FUNCTION_BLOCK FB_RobotAbsMove EXTENDS FB_ObjectBase_V2 IMPLEMENTS IBasicElement
VAR_INPUT
    Robot         : REFERENCE TO FB_FanucRobot_Basic_V2;
    LowerConveyor : REFERENCE TO FB_Motor;
    // Command   : ST_WareHouseWithRobotMove_Command;
    Info : st_AutoSixAxisAbsMoveParameter;
	Input :ST_InputTable;
    Stop : BOOL;
END_VAR
VAR_OUTPUT
    // Status : ST_WareHouseWithRobotMove_Status;
END_VAR
VAR
    _Abort       : BOOL;
    strStatus    : STRING;
    uiResumeStep : UINT;

    Area : E_RobotArea;
    UseA : BOOL;
    UseB : BOOL;

    Get                         : BOOL;
    tonTimeOut                  : TON;
	TON_DelayLowerCV			: TON;
    _UniqueErrorCode            : STRING;
    FirstSensorOfLowerConveyor  : BOOL;
    SecondSensorOfLowerConveyor : BOOL;

END_VAR

SUPER^.A10_StateControl();
A00_BasicUnits();
FirstSensorOfLowerConveyor := Input.bLowCV_BoxArrived_Sensor;
SecondSensorOfLowerConveyor := Input.bLowCV_2ndBoxGap_Sensor;

ACTION A00_BasicUnits:
tonTimeOut(PT:=T#60S);
TON_DelayLowerCV(PT:=T#1S);
ErrorID :=2200;
END_ACTION

METHOD M_CheckCommand : BOOL // True : Command is useful
VAR_INPUT
END_VAR
VAR
	
END_VAR
// Check command paremeter is correct


IF Info.A_Get <> Info.B_Get THEN
	strStatus:='Wrong command ,GetA not match to GetB';
	M_CheckCommand:=FALSE;
	RETURN;
ELSE		
	THIS^.Get :=Info.A_Get;
END_IF

IF Info.A_Area<> Info.B_Area THEN
	IF NOT(Info.A_Area=99 OR Info.B_Area=99) THEN
	strStatus:='Wrong command ,Area A not match to Area B';
	M_CheckCommand:=FALSE;
	RETURN;
END_IF
END_IF

IF Info.A_Area = 99 AND Info.B_Area = 99 THEN
	strStatus:='Wrong command ,Both Area are 99';
	M_CheckCommand:=FALSE;
	RETURN;
END_IF

CASE LREAL_TO_INT(Info.A_Area) OF
	1 : //Normal command : RoundBelt
		IF Info.A_Position<1 OR  Info.A_Position>3 THEN
			strStatus:='Wrong command ,Position A Not allow';
			M_CheckCommand:=FALSE;
			RETURN;	
		ELSE
			Area := E_RobotArea.RoundBelt;
			UseA :=TRUE	;	
		END_IF
		
	2:	//Buffer area
		IF Info.A_Position<1 OR  Info.A_Position>40 THEN
			strStatus:='Wrong command ,Position A Not allow';
			M_CheckCommand:=FALSE;
			RETURN;	
		ELSE
			Area := E_RobotArea.BufferArea;
			UseA :=TRUE	;	
		END_IF
	3: //Allocated/Empty conveyor
		IF Info.A_Position<1 OR  Info.A_Position>2 THEN
			strStatus:='Wrong command ,Position A Not allow';
			M_CheckCommand:=FALSE;
			RETURN;	
		ELSE
			Area := E_RobotArea.TransmitCV;
			UseA :=TRUE	;	
		END_IF
	5: //FeedIn/Out conveyor
		IF Info.A_Position<1 OR  Info.A_Position>3 THEN
			strStatus:='Wrong command ,Position A Not allow';
			M_CheckCommand:=FALSE;
			RETURN;	
		ELSIF Info.A_Position=3 AND Get THEN
			strStatus:='Wrong command ,Can Not Get box from FeedOut conveyor ';
			M_CheckCommand:=FALSE;
			RETURN;	
		ELSE
			Area := E_RobotArea.InOutConveyor;
			UseA :=TRUE	;	
		END_IF
	7: // PullOut conveyor
		IF Info.A_Position<1 OR  Info.A_Position>2 THEN
			strStatus:='Wrong command ,Position A Not allow';
			M_CheckCommand:=FALSE;
			RETURN;	
		ELSE
			Area := E_RobotArea.PullOutConveyor;
			UseA :=TRUE	;	
		END_IF
	
	99: //ClampA not use
		UseA :=FALSE;
	
	ELSE //Wrong command
		strStatus:='Wrong command ,Area_A not allow ';
		M_CheckCommand:=FALSE;
		RETURN;

END_CASE

CASE LREAL_TO_INT(Info.B_Area) OF
	1 : //Normal command : RoundBelt
		IF Info.B_Position<1 OR  Info.B_Position>3 THEN
			strStatus:='Wrong command ,Position B Not allow';
			M_CheckCommand:=FALSE;
			RETURN;	
		ELSE
			Area := E_RobotArea.RoundBelt;
			UseB :=TRUE	;	
		END_IF
		
	2:	
		IF Info.B_Position<1 OR  Info.B_Position>40 THEN
			strStatus:='Wrong command ,Position B Not allow';
			M_CheckCommand:=FALSE;
			RETURN;	
		ELSE
			Area := E_RobotArea.BufferArea;
			UseB :=TRUE	;	
		END_IF
	3:
		IF Info.B_Position<1 OR  Info.B_Position>2 THEN
			strStatus:='Wrong command ,Position B Not allow';
			M_CheckCommand:=FALSE;
			RETURN;	
		ELSE
			Area := E_RobotArea.TransmitCV;
			UseB :=TRUE	;	
		END_IF
	5:
		IF Info.B_Position<1 OR  Info.B_Position>3 THEN
			strStatus:='Wrong command ,Position B Not allow';
			M_CheckCommand:=FALSE;
			RETURN;	
		ELSE
			Area := E_RobotArea.InOutConveyor;
			UseB :=TRUE	;	
		END_IF
	7:
		IF Info.B_Position<1 OR  Info.B_Position>2 THEN
			strStatus:='Wrong command ,Position B Not allow';
			M_CheckCommand:=FALSE;
			RETURN;	
		ELSIF Info.B_Position=3 AND Get THEN
			strStatus:='Wrong command ,Can Not Get box from FeedOut conveyor ';
			M_CheckCommand:=FALSE;
			RETURN;	
		ELSE
			Area := E_RobotArea.PullOutConveyor;
			UseB :=TRUE	;	
		END_IF
	
	99: //ClampA not use
		UseB :=FALSE;
	
	ELSE //Wrong command
		strStatus:='Wrong command ,Area_B not allow ';
		M_CheckCommand:=FALSE;
		RETURN;

END_CASE


M_CheckCommand:=TRUE;
END_METHOD

METHOD M_CheckUnitsNotBusy : BOOL
VAR_INPUT
END_VAR
M_CheckUnitsNotBusy := true;
END_METHOD

METHOD M_CheckUnitsReady : BOOL
VAR_INPUT
END_VAR
M_CheckUnitsReady := true;
END_METHOD

METHOD  M_STATE_ABORTED
VAR_INPUT
END_VAR
ERROR :=TRUE;
Busy    := FALSE;
Aborted := TRUE;
Status := strStatus;
UniqueErrorCode:=_UniqueErrorCode;
IF NOT Execute THEN
	eSTATE:=STATE_RESETTING;
END_IF

IF Execute AND Reset THEN
	uiExecutingStep :=uiResumeStep;
	eSTATE:=STATE_EXECUTING;
END_IF
END_METHOD

METHOD  M_STATE_ABORTING
VAR_INPUT
END_VAR
CASE uiAbortingStep OF
	0 :
		uiAbortingStep:=9999;
	
	9999:	_AbortCompleted:=TRUE;
END_CASE

IF _AbortCompleted THEN	
	eSTATE :=STATE_ABORTED;
END_IF
END_METHOD

METHOD  M_STATE_DONE
VAR_INPUT
END_VAR
Busy := FALSE;
Done := TRUE;
IF NOT Execute THEN
    eState := STATE_RESETTING;
END_IF
END_METHOD

METHOD  M_STATE_DORMANT
VAR_INPUT
END_VAR
// Clear FB output
Busy            := FALSE;
Done            := FALSE;
Aborted         := FALSE;
Error           := FALSE;
ErrorID         := 0;
Status          := '';
_ResetCompleted := FALSE;
_Error          := FALSE;
_Executed       := FALSE;

tonTimeOut.IN:=FALSE;
TON_DelayLowerCV.IN := false;
strStatus :='No Error';
uiExecutingStep :=uiResettingStep :=uiResumeStep :=0;


// Wait Execute command
IF Execute THEN
    eState := STATE_EXECUTING;
END_IF
END_METHOD

METHOD  M_STATE_ERROR
VAR_INPUT
END_VAR
ERROR   :=TRUE;
Busy	:=FALSE;
Status := strStatus;
UniqueErrorCode:=_UniqueErrorCode;
ErrorID :=2200;
IF NOT Execute THEN	
eSTATE:=STATE_RESETTING;
END_IF
END_METHOD

METHOD  M_STATE_EXECUTING
VAR_INPUT
END_VAR
VAR_INST
    ActionMode       : E_ReloadRoundBoxAction;
	BoxReady_1st : BOOL;
	BoxReady_2nd : BOOL;
    CarrierReady_1st : BOOL;
    CarrierReady_2nd : BOOL;
    uiBothStep : UINT;
    uiSingleClampStep : UINT;	
	Area : E_RobotArea;
	Address_A : INT;
	Address_B : INT;
END_VAR
VAR
	WareHouse: INT;
END_VAR
// Set Busy active edit by johnson
Busy := TRUE;
IF THIS^.Stop THEN // Pending the timeout when Stop signal occur
	tonTimeout.IN :=FALSE;
END_IF
// Service Process
CASE uiExecutingStep OF
	0:
        // Clear variable
        ActionMode       := E_ReloadRoundBoxAction.Undefined;
        CarrierReady_1st := FALSE;
        CarrierReady_2nd := FALSE;
        uiBothStep := 0;
		uiSingleClampStep :=0;
		BoxReady_1st := 0;
		BoxReady_2nd := 0;
		tonTimeOut.IN:=FALSE;
        // Check command
        IF M_CheckCommand() THEN
            uiExecutingStep := 10;
		ELSE
			_Error:=TRUE;
        END_IF
    10:
        // Start process, check units first
        IF M_CheckUnitsReady() THEN
            uiExecutingStep := 20;
        END_IF
    20:
        // CHeck units not busy state
        IF M_CheckUnitsNotBusy() THEN
            uiExecutingStep := 1000;
        END_IF
   
	1000:   
			// Read   coordinate
			 Area := THIS^.Area;
 			 Address_A := LREAL_TO_INT(Info.A_Position);
			 Address_B := LREAL_TO_INT(Info.B_Position);
			 
			IF UseA AND NOT UseB THEN
				//Only clampA
				uiExecutingStep := 10000;
			ELSIF NOT UseA AND UseB THEN
				//Only ClampB 
				uiExecutingStep := 20000;
			ELSIF UseA AND UseB THEN
				//Both Clamps
				uiExecutingStep := 30000;		
			END_IF
       
    10000: // Only ClampA 
        IF NOT Robot._DI1.Done THEN
            
            
			CASE uiSingleClampStep OF
				
				0://
					IF Area= E_RobotArea.InOutConveyor AND Address_A=3 THEN
						uiSingleClampStep:=100;// Need to control feedout conveyor 
					ELSE
						uiSingleClampStep:=1000;	
					END_IF
				100:	//check the box is full 
					IF Input.bLowCV_Block2Detect_Sensor THEN 
						_Error := TRUE;
						strStatus :='LowerCV the box behind is full, please remove it';
					ELSE 
						uiSingleClampStep := 150;
					END_IF
				
				150:	//check the box not no the  sensor 
					IF  FirstSensorOfLowerConveyor OR  (NOT SecondSensorOfLowerConveyor) THEN
						LowerConveyor.M_MoveBackward();
						tonTimeOut.IN:=FALSE;;
						uiSingleClampStep:=200;
					ELSE 
						uiSingleClampStep := 1000;
					END_IF
					tonTimeOut.IN:=TRUE;
					IF tonTimeOut.Q=TRUE THEN
						strStatus :='Empty Conveyor timeout';
						_Error:=TRUE;
					END_IF
				200:
//					TON_DelayLowerCV.IN := TRUE;
//					IF TON_DelayLowerCV.Q THEN
//					LowerConveyor.M_MotorStop();
//					uiSingleClampStep:=300;
//					END_IF 
					IF Input.bLowCV_Block2Detect_Sensor THEN
						TON_DelayLowerCV.IN := TRUE;
					END_IF
					IF TON_DelayLowerCV.Q THEN
						LowerConveyor.M_MotorStop();
						uiSingleClampStep := 300;
					END_IF
									
				300:
					TON_DelayLowerCV.IN :=FALSE;
					IF 	LowerConveyor.InStopped THEN
						tonTimeOut.IN:=FALSE;
						uiSingleClampStep:=1000;
					END_IF
					tonTimeOut.IN:=TRUE;
					IF tonTimeOut.Q=TRUE THEN
						strStatus :='Stop Conveyor timeout';
						_Error:=TRUE;
					END_IF	
				1000:
						BoxReady_1st:=TRUE;
						uiSingleClampStep:=9999;
				9999: //Wait	
			END_CASE
			          		 
				  // Robot Abs move
           		 Robot.M_StartRobotAbsMove(GetBox:=Get,
											UseClampA:=UseA,
											UseClampB:=UseB,
											Area:=Area,
											ClampA_Address:=Address_A,
											ClampB_Address:=Address_B,
											BoxReady_1:=BoxReady_1st,
											BoxReady_2:=BoxReady_2nd);				  
		
        ELSE
            uiExecutingStep := 10080;
        END_IF
		
    10080:
        Robot.M_ResetRobotAbsMove(UseA,UseB); // Clear command and go to place box
		tonTimeOut.IN:=TRUE;
        IF NOT Robot._DI1.Done THEN
			tonTimeOut.IN:=FALSE;
            uiExecutingStep := 40000; 
        END_IF
    	IF tonTimeOut.Q=TRUE THEN
			strStatus :='Reset Robot timeout';
			_Error:=TRUE;
		END_IF
		
    
   20000: // Only ClampB
        IF NOT Robot._DI1.Done THEN
            			
			CASE uiSingleClampStep OF
				
				0://
					IF Area= E_RobotArea.InOutConveyor AND Address_B=3 THEN
						uiSingleClampStep:=100;// Need to control feedout conveyor 
					ELSE
						uiSingleClampStep:=1000;	
					END_IF
					
				100:	//check the box is full 
					IF Input.bLowCV_Block2Detect_Sensor THEN 
						_Error := TRUE;
						strStatus :='LowerCV the box behind is full, please remove it';
					ELSE 
						uiSingleClampStep := 150;
					END_IF
				
				150:	//check the box not no the  sensor 
					IF  FirstSensorOfLowerConveyor OR  (NOT SecondSensorOfLowerConveyor) THEN
						LowerConveyor.M_MoveBackward();
						tonTimeOut.IN:=FALSE;;
						uiSingleClampStep:=200;
					ELSE
						uiSingleClampStep := 1000;
					END_IF
					tonTimeOut.IN:=TRUE;
					IF tonTimeOut.Q=TRUE THEN
						strStatus :='Empty Conveyor timeout';
						_Error:=TRUE;
					END_IF
				200:
//					TON_DelayLowerCV.IN := TRUE;
//					IF TON_DelayLowerCV.Q THEN
//					LowerConveyor.M_MotorStop();
//					uiSingleClampStep:=300;
//					END_IF 
					IF Input.bLowCV_Block2Detect_Sensor THEN
						TON_DelayLowerCV.IN := TRUE;
					END_IF
					IF TON_DelayLowerCV.Q THEN
						LowerConveyor.M_MotorStop();
						uiSingleClampStep := 300;
					END_IF
									
				300:
					TON_DelayLowerCV.IN :=FALSE;
					IF 	LowerConveyor.InStopped THEN
						tonTimeOut.IN:=FALSE;
						uiSingleClampStep:=1000;
					END_IF
					tonTimeOut.IN:=TRUE;
					IF tonTimeOut.Q=TRUE THEN
						strStatus :='Stop Conveyor timeout';
						_Error:=TRUE;
					END_IF	
				1000:
						BoxReady_2nd:=TRUE;
						uiSingleClampStep:=9999;
				9999: //Wait			
			END_CASE
			          		 
				  // Robot Abs move
           		 Robot.M_StartRobotAbsMove( GetBox:=Get,
											UseClampA:=UseA,
											UseClampB:=UseB,
											Area:=Area,
											ClampA_Address:=Address_A,
											ClampB_Address:=Address_B,
											BoxReady_1:=BoxReady_1st,
											BoxReady_2:=BoxReady_2nd);	
        ELSE
            uiExecutingStep := 20080;
        END_IF
		
    20080:
       Robot.M_ResetRobotAbsMove(UseA,UseB);; // Clear command 

        IF NOT Robot._DI1.Done THEN
            uiExecutingStep := 40000; 
        END_IF
		tonTimeOut.IN:=TRUE;
		IF tonTimeOut.Q=TRUE THEN
			strStatus :='Reset Robot timeout';
			_Error:=TRUE;
		END_IF	
    30000: // Both Clamps
        		
		
		  CASE uiBothStep OF
           		0://	
					BoxReady_1st := FALSE;
					BoxReady_2nd := FALSE;
					IF Area= E_RobotArea.InOutConveyor AND Address_A=3 THEN
						uiBothStep:=100;// Need to control feedout conveyor 
					ELSE
						uiBothStep:=1000;	
					END_IF
					
				100:	//check the box is full 
					IF Input.bLowCV_Block2Detect_Sensor THEN 
						_Error := TRUE;
						strStatus :='LowerCV the box behind is full, please remove it';
					ELSE 
						uiBothStep := 200;
					END_IF
				
				200:	//check the box not no the  sensor 
					IF  FirstSensorOfLowerConveyor OR  (NOT SecondSensorOfLowerConveyor) THEN
						LowerConveyor.M_MoveBackward();
						tonTimeOut.IN:=FALSE;;
						uiBothStep:=300;
					ELSE
						uiBothStep := 1000;
					END_IF
					tonTimeOut.IN:=TRUE;
					IF tonTimeOut.Q=TRUE THEN
						strStatus :='Empty Conveyor timeout';
						_Error:=TRUE;
					END_IF
				300:
					IF Input.bLowCV_Block2Detect_Sensor THEN
						TON_DelayLowerCV.IN := TRUE;
					END_IF
					IF TON_DelayLowerCV.Q THEN
						LowerConveyor.M_MotorStop();
						uiBothStep := 400;
					END_IF
								
				400:
					TON_DelayLowerCV.IN :=FALSE;
					IF 	LowerConveyor.InStopped THEN
						tonTimeOut.IN:=FALSE;
						uiBothStep:=1000;
					END_IF
					tonTimeOut.IN:=TRUE;
					IF tonTimeOut.Q=TRUE THEN
						strStatus :='Stop Robot timeout';
						_Error:=TRUE;
					END_IF		
				1000:
						BoxReady_1st:=TRUE;
						uiBothStep:=2000;
						
				2000:
						IF Robot._DI1.Notification THEN
							uiBothStep:=3000;
						END_IF
				3000:
					
					IF Area= E_RobotArea.InOutConveyor AND Address_B=3 THEN
						uiBothStep:=3100;// Need to control feedout conveyor 
					ELSE
						uiBothStep:=9000;	
					END_IF
					
				3100:
					IF Input.bLowCV_Block2Detect_Sensor THEN 
						_Error := TRUE;
						strStatus :='LowerCV the box behind is full, please remove it';
					ELSE 
						uiBothStep := 3200;
					END_IF
				
				3200:	
					IF FirstSensorOfLowerConveyor OR (NOT SecondSensorOfLowerConveyor) THEN
						LowerConveyor.M_MoveBackward();
						tonTimeOut.IN:=FALSE;
						uiBothStep := 3300;
					ELSE 
						uiBothStep := 9000;
					END_IF
					tonTimeOut.IN:=TRUE;
					IF tonTimeOut.Q=TRUE THEN
						strStatus :='Empty Robot timeout';
						_Error:=TRUE;
					END_IF	
				3300:
					IF Input.bLowCV_Block2Detect_Sensor THEN
						TON_DelayLowerCV.IN := TRUE;
					END_IF
					IF TON_DelayLowerCV.Q THEN
						LowerConveyor.M_MotorStop();
						uiBothStep := 3400;
					END_IF
				
				3400:
					TON_DelayLowerCV.IN :=FALSE;
					IF 	LowerConveyor.InStopped THEN
						tonTimeOut.IN:=FALSE;
						uiBothStep:=9000;
					END_IF
					tonTimeOut.IN:=TRUE;
					IF tonTimeOut.Q=TRUE THEN
						strStatus :='Stop Robot timeout';
						_Error:=TRUE;
					END_IF		
				9000:
						BoxReady_2nd:=TRUE;
						uiBothStep:=9999;
				
				9999: //Wait		
        // wait reset
        END_CASE

       	  // Robot Abs move
           		 Robot.M_StartRobotAbsMove( GetBox:=Get,
											UseClampA:=UseA,
											UseClampB:=UseB,
											Area:=Area,
											ClampA_Address:=Address_A,
											ClampB_Address:=Address_B,
											BoxReady_1:=BoxReady_1st,
											BoxReady_2:=BoxReady_2nd);	
		
		
        IF Robot._DI1.Done THEN
            uiExecutingStep := 30080;
        END_IF
		
    30080: // Check robot command is clear
        
        Robot.M_ResetRobotAbsMove(UseA,UseB);

        IF NOT Robot._DI1.Done THEN
			tonTimeOut.IN:=FALSE;
            uiExecutingStep := 40000; // go to place step
        END_IF    
   		//tonTimeOut.IN:=TRUE;
		IF tonTimeOut.Q=TRUE THEN
			strStatus :='Stop Robot timeout';
			_Error:=TRUE;
		END_IF

	40000:  //check the box is full ## Edit BY MIN 20250416
			 
			IF Input.bLowCV_Block2Detect_Sensor THEN 
				_Error := TRUE;
				strStatus :='LowerCV the box behind is full, please remove it';
			ELSE 
				uiExecutingStep := 40100;
			END_IF	
	
	40100:
			IF  FirstSensorOfLowerConveyor OR (NOT SecondSensorOfLowerConveyor) THEN
				tonTimeOut.IN:=FALSE;
				LowerConveyor.M_MoveBackward();
				uiExecutingStep:=40200;
			ELSE
				uiExecutingStep:=99000;
			END_IF
			tonTimeOut.IN:=TRUE;
			IF tonTimeOut.Q=TRUE THEN
				strStatus :='Lowerconveyor Reverse timeout';
				_Error:=TRUE;
			END_IF	
			
	40200:
			tonTimeOut.IN:=FALSE;
			IF Input.bLowCV_Block2Detect_Sensor THEN
				TON_DelayLowerCV.IN := TRUE;
			END_IF
			IF TON_DelayLowerCV.Q THEN
				LowerConveyor.M_MotorStop();
				uiExecutingStep := 40300;
			END_IF
			
	40300:
			IF LowerConveyor.InStopped THEN
					IF NOT (FirstSensorOfLowerConveyor) AND  SecondSensorOfLowerConveyor THEN
						uiExecutingStep := 99000;
					ELSE
						_Error := TRUE;
						strStatus := 'LowerCV the box Behind is full ,please remove it ';
					END_IF	
			END_IF
			
			tonTimeOut.IN:=TRUE;
			IF tonTimeOut.Q=TRUE THEN
				strStatus :='Lowerconveyor Reverse Stop timeout';
				_Error:=TRUE;
			END_IF
			
			
   
    99000: // process done
			TON_DelayLowerCV.IN :=FALSE;
                Status    := 'Process completed';
        		_Executed := TRUE;
END_CASE
IF _Executed THEN
    eState := STATE_DONE;
ELSIF _Error THEN
	//(iErrorID := ErrorID,UinqueErrorCode=>_UniqueErrorCode);
    eState := STATE_ERROR;
ELSIF NOT Execute THEN
    eState := STATE_RESETTING;
END_IF
IF _Abort OR Abort THEN
	//FUN_UniqueErrorCodeGenerator(iErrorID := ErrorID,UinqueErrorCode=>_UniqueErrorCode);
	eSTATE:=STATE_ABORTING;
END_IF
END_METHOD

METHOD  M_STATE_RESETTING
VAR_INPUT
END_VAR
Error :=FALSE;
Done :=FALSE;
Busy := FALSE;


CASE uiResettingStep OF
	
	0:
		tonTimeOut.IN:=FALSE;
		TON_DelayLowerCV.IN := false;
		Robot.M_ResetAllCommand();
		Robot.M_ResetRobotAbsMove(TRUE,TRUE);
		uiResettingStep:=100;
		
	100:
	
		LowerConveyor.M_MotorStop();	
		uiResettingStep:=9999;
	9999:
		_ResetCompleted:=TRUE;
END_CASE
IF _ResetCompleted THEN
	eSTATE:=STATE_DORMANT;
END_IF
END_METHOD

END_FUNCTION_BLOCK

(* stored: Version 1.1.0.1, ProductVersion 3.1.4024.13
   POU FB_RobotAbsMove: Id {1ad501e0-b8bd-4d34-ac88-449f5666c9d1}, SpecialFunc None
   Folder Method: Id {4e56b499-26f7-43b9-9264-4d7f7db7a928}
   Folder State: Id {5851a20e-bfcb-4cc2-912a-b5cbbc3cf000}
   Action A00_BasicUnits: Id {5e2200d6-cccc-47bc-9cfb-02eb0dfbdf3e}
   Method M_CheckCommand: Id {10bc46a1-7ff8-4785-9eab-11ce7e3f6c17}
   Method M_CheckUnitsNotBusy: Id {8a0f2757-7cb3-418a-a77c-825750b924b7}
   Method M_CheckUnitsReady: Id {503f7e8c-48c4-4fca-b01a-aa77c30f2f19}
   Method M_STATE_ABORTED: Id {b8446965-6d28-42df-b8d6-7f41eeaa5288}
   Method M_STATE_ABORTING: Id {20f5ec62-eff2-48bd-b5a7-a5ff1a274748}
   Method M_STATE_DONE: Id {6e587ace-b076-4d1f-9be0-f15d02920a20}
   Method M_STATE_DORMANT: Id {7366a93a-51a7-4755-bc6e-6f7e4cb042b0}
   Method M_STATE_ERROR: Id {36940727-e798-4f5b-8181-2b4817b4ed57}
   Method M_STATE_EXECUTING: Id {d73533ac-5232-410b-9b0d-37327b450aef}
   Method M_STATE_RESETTING: Id {d89f63ec-10d4-451a-b28a-23ea9dbf81fb} *)
